RoboDK station: test.rdk

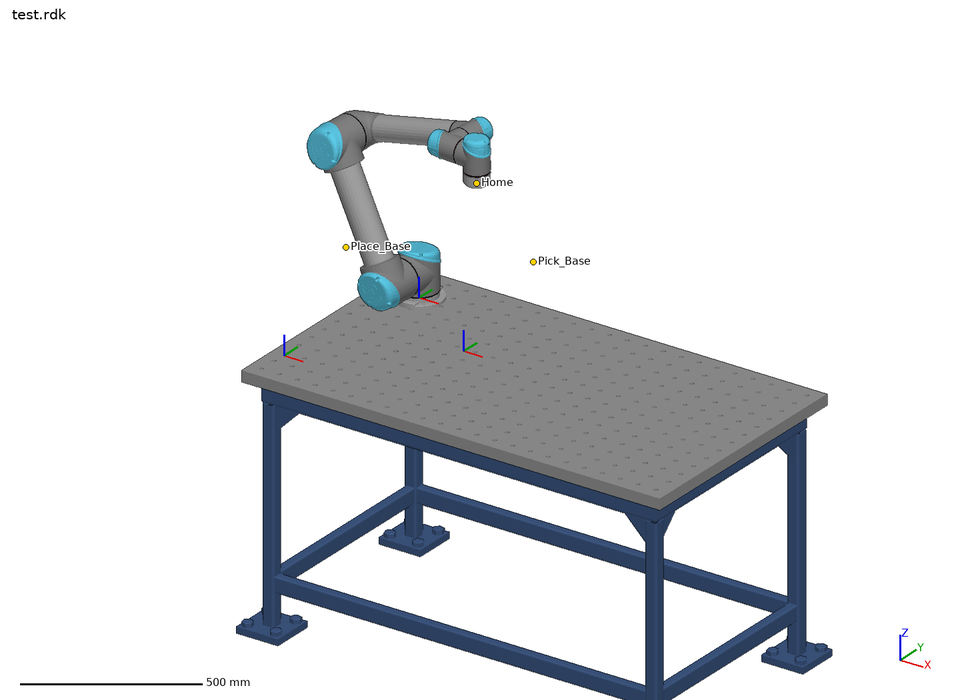
[picture v0: the station drawn from its stored meshes, robots at their saved joint values, targets as dots, program paths as lines]
Station test (saved by RoboDK 5.5.4). Poses are relative to the parent item; angles as X-Y-Z fixed-axis rotations.
  - frame UR5 Base at (0, 0, 0) mm
    - robot UR5: 6 axes
        modified DH rows (alpha deg, a mm, theta deg, d mm): 0, 0, 0, 89.2; 90, 0, 180, 0; 0, 425, 0, 0; 0, 392, 0, 109.3; -90, 0, 0, 94.75; 90, 0, 0, 82.5
        joint limits [-360, -360, -360, -360, -360, -360] to [360, 360, 360, 360, 360, 360]; home [0, -90, -90, 0, 90, 0]; saved at [-3.93, -64.188, -102.509, -103.304, 90, -3.93]
  - frame Wordl at (0, 0, 0) mm
    - object Table 1400x800x800mm at (200, -250, 0) mm, size 1420 x 820 x 800 mm, geometry from Table-1400x800x800mm.sld
    - target Home (Cartesian target) at (283, -129, 479.5) mm, rotated rx -180 ry 0 rz -90 deg; joints [-3.93, -64.188, -102.509, -103.304, 90, -3.93] of UR5
    - target Place_Base (Cartesian target) at (7.75, -358.5, 300) mm, rotated rx -180 ry 0 rz -90 deg; joints [-71.015, -72.331, -124.217, -73.452, 90, -71.015] of UR5
    - target Pick_Base (Cartesian target) at (414.5, -44.5, 242) mm, rotated rx -180 ry 0 rz -90 deg; joints [9.072, -85.094, -123.589, -61.317, 90.001, 9.072] of UR5
  - frame Pick_Mat at (291.34, -203.01, 0) mm
  - frame Build_plate at (-95.4, -507.4, 0) mm
